// TIA Portal project "conveyer belt system V5.1" (V19)

(* hardware
DEVICE "S71500/ET200MP-Station_1"  S7-1500 station
   slot 0: "Profilschiene_0"  6ES7 590-1***0-0AA0
   slot 1: "PLC_1"  CPU 1511-1 PN  6ES7 511-1AK00-0AB0  V1.8
   slot 2: "AI 8xU/I/RTD/TC ST_1"  AI 8xU/I/RTD/TC ST  6ES7 531-7KF00-0AB0  V2.0
   slot 3: "AI 8xU/I/RTD/TC ST_2"  AI 8xU/I/RTD/TC ST  6ES7 531-7KF00-0AB0  V2.0
   slot 4: "AI 8xU/I/RTD/TC ST_3"  AI 8xU/I/RTD/TC ST  6ES7 531-7KF00-0AB0  V2.0
   slot 5: "AI 8xU/I/RTD/TC ST_4"  AI 8xU/I/RTD/TC ST  6ES7 531-7KF00-0AB0  V2.0
   slot 6: "DI 16x24VDC BA_1"  DI 16x24VDC BA  6ES7 521-1BH10-0AA0  V1.0
*)

// ===== PLC "PLC_1"  CPU 1511-1 PN =====

VAR_GLOBAL   // PLC tag table "Standard-Variablentabelle"
   "Tag_1" AT %I1000.0 : Bool;
   "Tag_2" AT %Q1000.0 : Bool;
   "Tag_3" AT %I1000.1 : Bool;
END_VAR

VAR_GLOBAL   // PLC tag table "control panel"
   "start button" AT %I0.0 : Bool;
   "reset button" AT %I0.1 : Bool;
   "stop button" AT %I0.2 : Bool;
   "emergency stop" AT %I0.3 : Bool;
   "start button light" AT %Q0.0 : Bool;
   "reset button light" AT %Q0.1 : Bool;
   "stop button light" AT %Q0.2 : Bool;
   "system start" AT %Q0.3 : Bool;
   "system fault" AT %Q0.4 : Bool;
   "system stop" AT %Q0.5 : Bool;
   "sensor start" AT %I0.7 : Bool;
   "low power mode" AT %I0.4 : Bool;
END_VAR

VAR_GLOBAL   // PLC tag table "conveyor 0"
   "motor +(0)" AT %Q3.7 : Bool;
   "motor -(0)" AT %Q3.6 : Bool;
   "encoder A(0)" AT %I3.7 : Bool;
   "encoder B(0)" AT %I3.6 : Bool;
   "sensor(0)" AT %I5.7 : Bool;
END_VAR

VAR_GLOBAL   // PLC tag table "conveyor 1"
   "motor +(1)" AT %Q3.5 : Bool;
   "motor -(1)" AT %Q3.4 : Bool;
   "encoder A(1)" AT %I3.5 : Bool;
   "encoder B(1)" AT %I3.4 : Bool;
   "sensor(1)" AT %I5.6 : Bool;
END_VAR

VAR_GLOBAL   // PLC tag table "conveyor 2"
   "motor +(2)" AT %Q3.3 : Bool;
   "motor -(2)" AT %Q3.2 : Bool;
   "encoder A(2)" AT %I3.3 : Bool;
   "encoder B(2)" AT %I3.2 : Bool;
   "sensor(2)" AT %I5.5 : Bool;
END_VAR

VAR_GLOBAL   // PLC tag table "system state"
   "start 0" AT %M0.0 : Bool;
   "start 1" AT %M0.1 : Bool;
   "conveyor 0 running" AT %M10.0 : Bool;
   "conveyor 1 running" AT %M10.1 : Bool;
   "conveyor 2 running" AT %M10.2 : Bool;
   "sensor 0 memory" AT %M20.0 : Bool;
   "sensor 1 memory" AT %M20.1 : Bool;
   "sensor 2 memory" AT %M20.2 : Bool;
   "sensor start memory" AT %M30.0 : Bool;
   "all conveyors running" AT %M0.2 : Bool;
   "system start/stop memory" AT %M0.4 : Bool;
   "conveyors running" AT %M0.3 : Bool;
   "sensor 3 memory" AT %M20.3 : Bool;
   "sensor 4 memory" AT %M20.4 : Bool;
   "sensor 5 memory" AT %M20.5 : Bool;
   "sensor 6 memory" AT %M20.6 : Bool;
   "conveyor 3 running" AT %M10.3 : Bool;
   "conveyor 4 running" AT %M10.4 : Bool;
   "conveyor 5 running" AT %M10.5 : Bool;
   "conveyor 6 running" AT %M10.6 : Bool;
END_VAR

VAR_GLOBAL   // PLC tag table "conveyor 3"
   "motor +(3)" AT %Q3.1 : Bool;
   "motor -(3)" AT %Q3.0 : Bool;
   "encoder A(3)" AT %I3.1 : Bool;
   "encoder B(3)" AT %I3.0 : Bool;
   "sensor(3)" AT %I5.4 : Bool;
END_VAR

VAR_GLOBAL   // PLC tag table "conveyor 4"
   "motor +(4)" AT %Q2.7 : Bool;
   "motor -(4)" AT %Q2.6 : Bool;
   "encoder A(4)" AT %I2.7 : Bool;
   "encoder B(4)" AT %I2.6 : Bool;
   "sensor(4)" AT %I5.3 : Bool;
END_VAR

VAR_GLOBAL   // PLC tag table "conveyor 5"
   "motor +(5)" AT %Q2.5 : Bool;
   "motor -(5)" AT %Q2.4 : Bool;
   "encoder A(5)" AT %I2.5 : Bool;
   "encoder B(5)" AT %I2.4 : Bool;
   "sensor(5)" AT %I5.2 : Bool;
END_VAR

VAR_GLOBAL   // PLC tag table "conveyor 6"
   "motor +(6)" AT %Q2.3 : Bool;
   "motor -(6)" AT %Q2.2 : Bool;
   "encoder A(6)" AT %I2.3 : Bool;
   "encoder B(6)" AT %I2.2 : Bool;
   "sensor(6)" AT %I5.1 : Bool;
END_VAR

DATA_BLOCK "conveyor_0"   // DB1
{ S7_Optimized_Access := 'TRUE' }
VERSION : 0.1
// stored: InstanceOfName conveyor control
"conveyor control"
BEGIN
END_DATA_BLOCK

DATA_BLOCK "conveyor_2"   // DB3
{ S7_Optimized_Access := 'TRUE' }
VERSION : 0.1
// stored: InstanceOfName conveyor control
"conveyor control"
BEGIN
END_DATA_BLOCK

DATA_BLOCK "conveyor_1"   // DB5
{ S7_Optimized_Access := 'TRUE' }
VERSION : 0.1
// stored: InstanceOfName conveyor control
"conveyor control"
BEGIN
END_DATA_BLOCK

DATA_BLOCK "sensor control_0"   // DB8
{ S7_Optimized_Access := 'TRUE' }
VERSION : 0.1
// stored: InstanceOfName sensor control
"sensor control"
BEGIN
END_DATA_BLOCK

DATA_BLOCK "sensor control_1"   // DB9
{ S7_Optimized_Access := 'TRUE' }
VERSION : 0.1
// stored: InstanceOfName sensor control
"sensor control"
BEGIN
END_DATA_BLOCK

DATA_BLOCK "sensor control_2"   // DB10
{ S7_Optimized_Access := 'TRUE' }
VERSION : 0.1
// stored: InstanceOfName sensor control
"sensor control"
BEGIN
END_DATA_BLOCK

DATA_BLOCK "lamp control_DB"   // DB11
{ S7_Optimized_Access := 'TRUE' }
VERSION : 0.1
// stored: InstanceOfName lamp control
"lamp control"
BEGIN
END_DATA_BLOCK

DATA_BLOCK "start pulse"   // DB12
{ S7_Optimized_Access := 'TRUE' }
VERSION : 0.1
// stored: InstanceOfName pulse
"pulse"
BEGIN
END_DATA_BLOCK

DATA_BLOCK "stop pulse"   // DB13
{ S7_Optimized_Access := 'TRUE' }
VERSION : 0.1
// stored: InstanceOfName pulse
"pulse"
BEGIN
END_DATA_BLOCK

DATA_BLOCK "conveyor_3"   // DB15
{ S7_Optimized_Access := 'TRUE' }
VERSION : 0.1
// stored: InstanceOfName conveyor control
"conveyor control"
BEGIN
END_DATA_BLOCK

DATA_BLOCK "conveyor_4"   // DB17
{ S7_Optimized_Access := 'TRUE' }
VERSION : 0.1
// stored: InstanceOfName conveyor control
"conveyor control"
BEGIN
END_DATA_BLOCK

DATA_BLOCK "conveyor_5"   // DB19
{ S7_Optimized_Access := 'TRUE' }
VERSION : 0.1
// stored: InstanceOfName conveyor control
"conveyor control"
BEGIN
END_DATA_BLOCK

DATA_BLOCK "conveyor_6"   // DB21
{ S7_Optimized_Access := 'TRUE' }
VERSION : 0.1
// stored: InstanceOfName conveyor control
"conveyor control"
BEGIN
END_DATA_BLOCK

DATA_BLOCK "sensor control_3"   // DB22
{ S7_Optimized_Access := 'TRUE' }
VERSION : 0.1
// stored: InstanceOfName sensor control
"sensor control"
BEGIN
END_DATA_BLOCK

DATA_BLOCK "sensor control_4"   // DB23
{ S7_Optimized_Access := 'TRUE' }
VERSION : 0.1
// stored: InstanceOfName sensor control
"sensor control"
BEGIN
END_DATA_BLOCK

DATA_BLOCK "sensor control_5"   // DB24
{ S7_Optimized_Access := 'TRUE' }
VERSION : 0.1
// stored: InstanceOfName sensor control
"sensor control"
BEGIN
END_DATA_BLOCK

DATA_BLOCK "sensor control_6"   // DB25
{ S7_Optimized_Access := 'TRUE' }
VERSION : 0.1
// stored: InstanceOfName sensor control
"sensor control"
BEGIN
END_DATA_BLOCK

DATA_BLOCK "standard parameters"   // DB26
{ S7_Optimized_Access := 'TRUE' }
VERSION : 0.1
   VAR
      "2 meter belt clearance delay" : Time := T#4S;
      "4 meter belt clearance delay" : Time := T#8S;
      "6 meter belt clearance delay" : Time := T#12S;
      "curved belt clearance delay" : Time := T#4S;
   END_VAR
BEGIN
END_DATA_BLOCK

DATA_BLOCK "system state"   // DB27
{ S7_Optimized_Access := 'TRUE' }
VERSION : 0.1
   VAR
      "start 0" : Bool;
      "start 1" : Bool;
      "all conveyors running" : Bool;
      "conveyors running" : Bool;
      "system start/stop memory" : Bool;
      "conveyor 0 running" : Bool;
      "conveyor 1 running" : Bool;
      "conveyor 2 running" : Bool;
      "conveyor 3 running" : Bool;
      "conveyor 4 running" : Bool;
      "conveyor 5 running" : Bool;
      "conveyor 6 running" : Bool;
      "sensor 0 memory" : Bool;
      "sensor 1 memory" : Bool;
      "sensor 2 memory" : Bool;
      "sensor 3 memory" : Bool;
      "sensor 4 memory" : Bool;
      "sensor 5 memory" : Bool;
      "sensor 6 memory" : Bool;
      "sensor start memory" : Bool;
   END_VAR
BEGIN
END_DATA_BLOCK

// folder: System blocks/Program resources

DATA_BLOCK "conveyor start delay"   // DB2
{ S7_Optimized_Access := 'TRUE' }
AUTHOR : Simatic
FAMILY : IEC
NAME : IEC_TMR
VERSION : 1.0
// stored: InstanceOfName IEC_TIMER
"IEC_TIMER"
BEGIN
END_DATA_BLOCK

DATA_BLOCK "delay 1"   // DB4
{ S7_Optimized_Access := 'TRUE' }
AUTHOR : Simatic
FAMILY : IEC
NAME : IEC_TMR
VERSION : 1.0
// stored: InstanceOfName IEC_TIMER
"IEC_TIMER"
BEGIN
END_DATA_BLOCK

DATA_BLOCK "delay 2"   // DB6
{ S7_Optimized_Access := 'TRUE' }
AUTHOR : Simatic
FAMILY : IEC
NAME : IEC_TMR
VERSION : 1.0
// stored: InstanceOfName IEC_TIMER
"IEC_TIMER"
BEGIN
END_DATA_BLOCK

DATA_BLOCK "delay 0"   // DB7
{ S7_Optimized_Access := 'TRUE' }
AUTHOR : Simatic
FAMILY : IEC
NAME : IEC_TMR
VERSION : 1.0
// stored: InstanceOfName IEC_TIMER
"IEC_TIMER"
BEGIN
END_DATA_BLOCK

DATA_BLOCK "delay 3"   // DB14
{ S7_Optimized_Access := 'TRUE' }
AUTHOR : Simatic
FAMILY : IEC
NAME : IEC_TMR
VERSION : 1.0
// stored: InstanceOfName IEC_TIMER
"IEC_TIMER"
BEGIN
END_DATA_BLOCK

DATA_BLOCK "delay 4"   // DB16
{ S7_Optimized_Access := 'TRUE' }
AUTHOR : Simatic
FAMILY : IEC
NAME : IEC_TMR
VERSION : 1.0
// stored: InstanceOfName IEC_TIMER
"IEC_TIMER"
BEGIN
END_DATA_BLOCK

DATA_BLOCK "delay 5"   // DB18
{ S7_Optimized_Access := 'TRUE' }
AUTHOR : Simatic
FAMILY : IEC
NAME : IEC_TMR
VERSION : 1.0
// stored: InstanceOfName IEC_TIMER
"IEC_TIMER"
BEGIN
END_DATA_BLOCK

DATA_BLOCK "delay 6"   // DB20
{ S7_Optimized_Access := 'TRUE' }
AUTHOR : Simatic
FAMILY : IEC
NAME : IEC_TMR
VERSION : 1.0
// stored: InstanceOfName IEC_TIMER
"IEC_TIMER"
BEGIN
END_DATA_BLOCK

// folder: (top level)

FUNCTION_BLOCK "conveyor control"   // FB1, FBD
{ S7_Optimized_Access := 'TRUE' }
VERSION : 0.1
   VAR_INPUT
      enable : Bool;
      "encoder A" : Bool;
      "encoder B" : Bool;
   END_VAR
   VAR_OUTPUT
      "running feedback" : Bool;
      "motor +" : Bool;
      "motor -" : Bool;
   END_VAR
   VAR
      "encoder buffer" : TOF_TIME;
      "encoder A edge" : R_TRIG;
      "encoder B edge" : R_TRIG;
   END_VAR
BEGIN

REGION Network 1
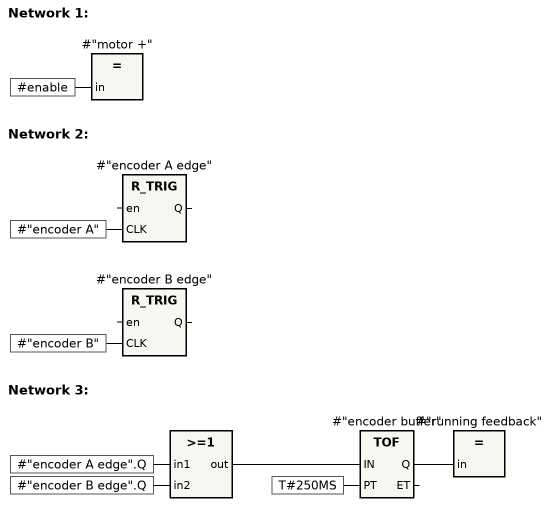
   #"motor +" := #enable;
END_REGION

REGION Network 2
   #"encoder A edge"(CLK := #"encoder A");   // R_TRIG
   #"encoder B edge"(CLK := #"encoder B");   // R_TRIG
END_REGION

REGION Network 3
   #"encoder buffer"(IN := #"encoder A edge".Q OR #"encoder B edge".Q, PT := T#250MS);   // TOF
   #"running feedback" := #"encoder buffer".Q;
END_REGION
END_FUNCTION_BLOCK

FUNCTION_BLOCK "sensor control"   // FB2, FBD
{ S7_Optimized_Access := 'TRUE' }
VERSION : 0.1
   VAR_INPUT
      "clearance delay" : Time;
      sensor : Bool;
      "preceding sensor" : Bool;
   END_VAR
   VAR_OUTPUT
      "motor +" : Bool;
   END_VAR
   VAR
      "clearance timer off" : TOF_TIME;
      "clearance timer on" : TOF_TIME;
      "clearance delay off" : TOF_TIME;
      "clearance delay on" : TON_TIME;
      "sensor memory" : Bool;
   END_VAR
BEGIN

REGION Network 1
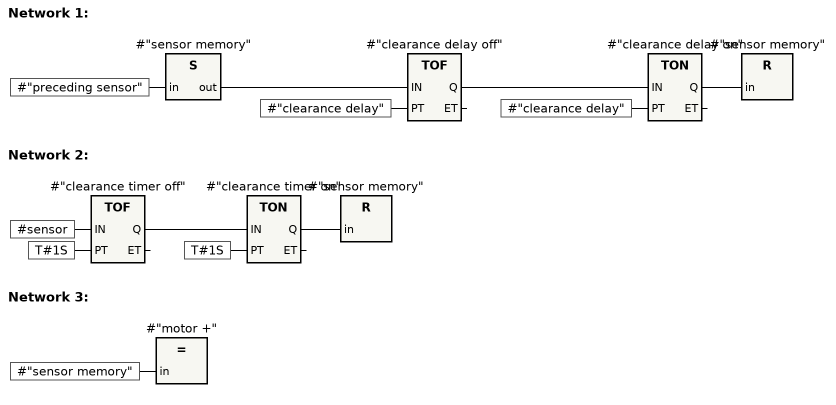
   IF #"preceding sensor" THEN #"sensor memory" := TRUE; END_IF;
   #"clearance delay off"(IN := #"preceding sensor", PT := #"clearance delay");   // TOF
   #"clearance delay on"(IN := #"clearance delay off".Q, PT := #"clearance delay");   // TON
   IF #"clearance delay on".Q THEN #"sensor memory" := FALSE; END_IF;
END_REGION

REGION Network 2
   #"clearance timer off"(IN := #sensor, PT := T#1S);   // TOF
   #"clearance timer on"(IN := #"clearance timer off".Q, PT := T#1S);   // TON
   IF #"clearance timer on".Q THEN #"sensor memory" := FALSE; END_IF;
END_REGION

REGION Network 3
   #"motor +" := #"sensor memory";
END_REGION
END_FUNCTION_BLOCK

FUNCTION_BLOCK "lamp control"   // FB3, FBD
{ S7_Optimized_Access := 'TRUE' }
VERSION : 0.1
   VAR_INPUT
      "system start" : Bool;
      "system fault" : Bool;
      "system stop" : Bool;
   END_VAR
BEGIN

REGION Network 1
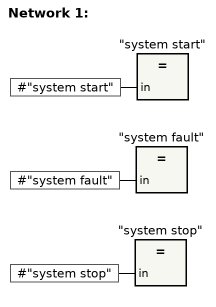
   "system start" := #"system start";
   "system fault" := #"system fault";
   "system stop" := #"system stop";
END_REGION
END_FUNCTION_BLOCK

FUNCTION_BLOCK "pulse"   // FB4, FBD
{ S7_Optimized_Access := 'TRUE' }
VERSION : 0.1
   VAR_INPUT
      enable : Bool;
      "pulse time" : Time;
   END_VAR
   VAR_OUTPUT
      "pulsing output" : Bool;
   END_VAR
   VAR
      "time delay bit" : Bool;
      IEC_Timer_0_Instance : TON_TIME;
      IEC_Timer_0_Instance_1 : TON_TIME;
   END_VAR
BEGIN

REGION Network 1
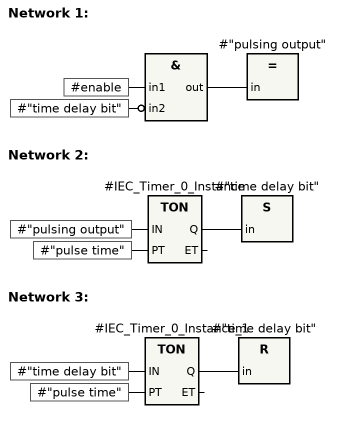
   #"pulsing output" := #enable AND NOT #"time delay bit";
END_REGION

REGION Network 2
   #IEC_Timer_0_Instance(IN := #"pulsing output", PT := #"pulse time");   // TON
   IF #IEC_Timer_0_Instance.Q THEN #"time delay bit" := TRUE; END_IF;
END_REGION

REGION Network 3
   #IEC_Timer_0_Instance_1(IN := #"time delay bit", PT := #"pulse time");   // TON
   IF #IEC_Timer_0_Instance_1.Q THEN #"time delay bit" := FALSE; END_IF;
END_REGION
END_FUNCTION_BLOCK

FUNCTION "default condition" : Void   // FC1, FBD
{ S7_Optimized_Access := 'TRUE' }
VERSION : 0.1
   VAR_TEMP   // added for the SCL form of the ladder/FBD networks
      _w1 : Bool;
      _w2 : Bool;
      _w3 : Bool;
   END_VAR
BEGIN

REGION Network 1: system start delay
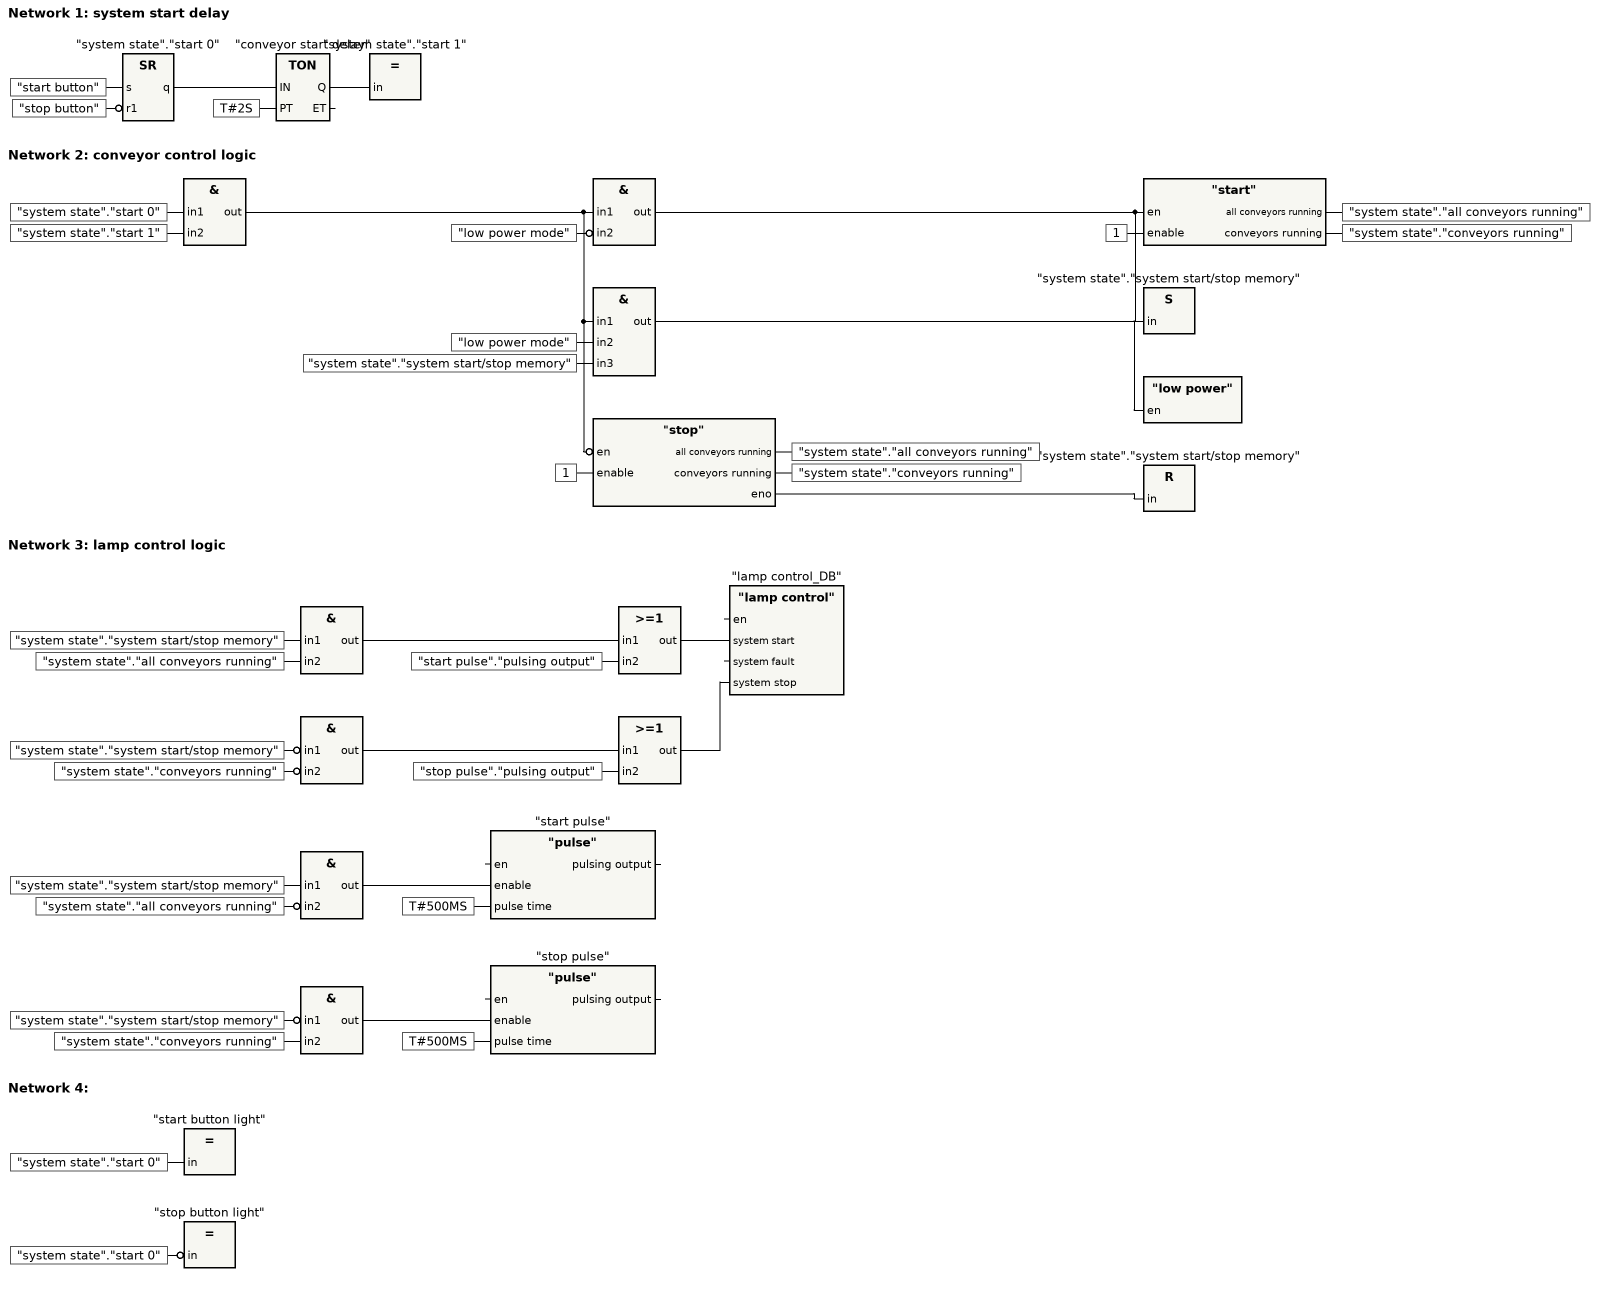
   IF "start button" THEN
       "system state"."start 0" := TRUE;   // SR flip-flop
   END_IF;
   IF NOT "stop button" THEN "system state"."start 0" := FALSE; END_IF;
   "conveyor start delay".TON(IN := "system state"."start 0", PT := T#2S);
   "system state"."start 1" := "conveyor start delay".Q;
END_REGION

REGION Network 2: conveyor control logic
   #_w1 := "system state"."start 0" AND "system state"."start 1";
   #_w2 := #_w1 AND NOT "low power mode";
   IF #_w2 THEN
       "start"(enable := 1,
               "all conveyors running" => "system state"."all conveyors running",
               "conveyors running" => "system state"."conveyors running");
       "system state"."system start/stop memory" := TRUE;
   END_IF;
   IF #_w1 AND "low power mode" AND "system state"."system start/stop memory" THEN "low power"(); END_IF;
   "stop"(EN := NOT #_w1,
          enable := 1,
          "all conveyors running" => "system state"."all conveyors running",
          "conveyors running" => "system state"."conveyors running",
          ENO => #_w3);
   IF #_w3 THEN "system state"."system start/stop memory" := FALSE; END_IF;
END_REGION

REGION Network 3: lamp control logic
   "lamp control_DB"("system start" := ("system state"."system start/stop memory" AND "system state"."all conveyors running") OR "start pulse"."pulsing output",   // "lamp control"
                     "system stop" := (NOT "system state"."system start/stop memory" AND NOT "system state"."conveyors running") OR "stop pulse"."pulsing output");
   "start pulse"(enable := "system state"."system start/stop memory" AND NOT "system state"."all conveyors running",   // "pulse"
                 "pulse time" := T#500MS);
   "stop pulse"(enable := NOT "system state"."system start/stop memory" AND "system state"."conveyors running",   // "pulse"
                "pulse time" := T#500MS);
END_REGION

REGION Network 4
   "start button light" := "system state"."start 0";
   "stop button light" := NOT "system state"."start 0";
END_REGION
END_FUNCTION

FUNCTION "start" : Void   // FC2, FBD
{ S7_Optimized_Access := 'TRUE' }
VERSION : 0.1
   VAR_INPUT
      enable : Bool;
   END_VAR
   VAR_OUTPUT
      "all conveyors running" : Bool;
      "conveyors running" : Bool;
   END_VAR
BEGIN

REGION Network 1
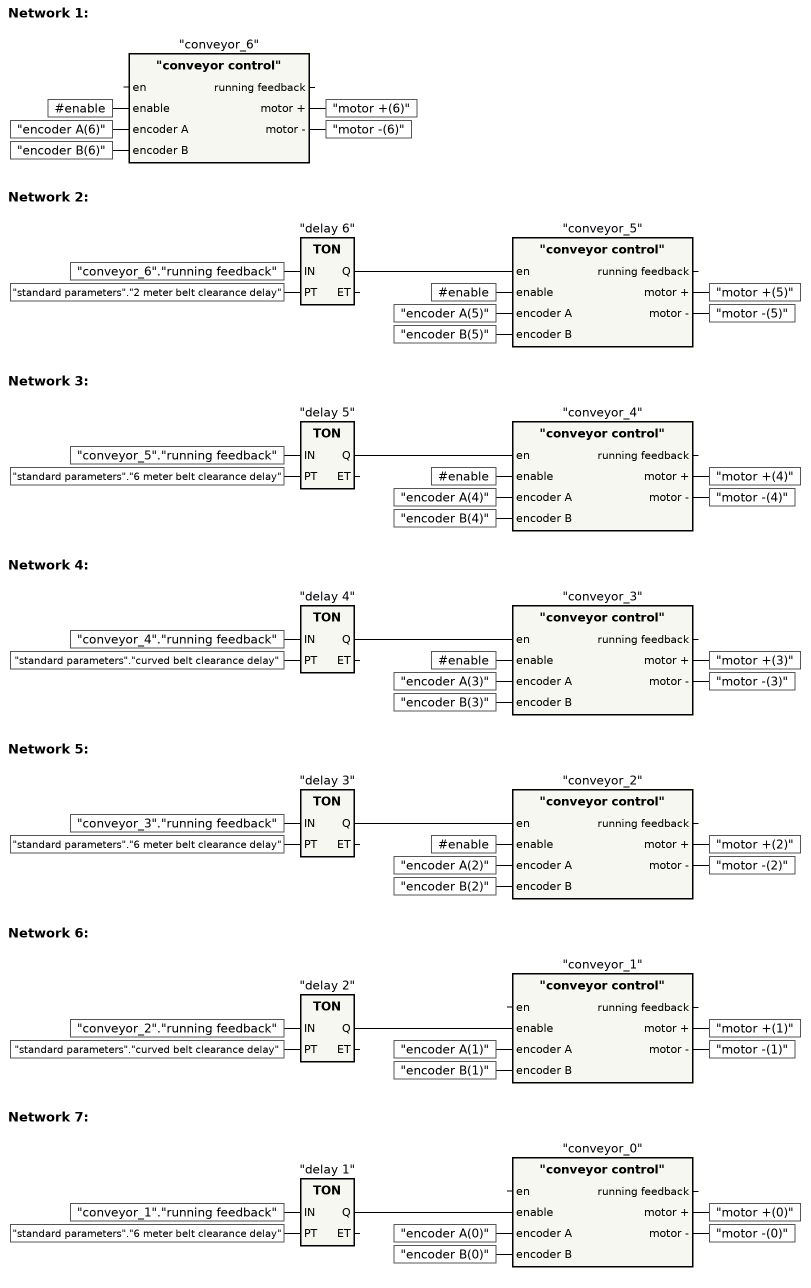
   "conveyor_6"(enable := #enable,   // "conveyor control"
                "encoder A" := "encoder A(6)",
                "encoder B" := "encoder B(6)",
                "motor +" => "motor +(6)",
                "motor -" => "motor -(6)");
END_REGION

REGION Network 2
   "delay 6".TON(IN := "conveyor_6"."running feedback",
                 PT := "standard parameters"."2 meter belt clearance delay");
   IF "delay 6".Q THEN
       "conveyor_5"(enable := #enable,   // "conveyor control"
                    "encoder A" := "encoder A(5)",
                    "encoder B" := "encoder B(5)",
                    "motor +" => "motor +(5)",
                    "motor -" => "motor -(5)");
   END_IF;
END_REGION

REGION Network 3
   "delay 5".TON(IN := "conveyor_5"."running feedback",
                 PT := "standard parameters"."6 meter belt clearance delay");
   IF "delay 5".Q THEN
       "conveyor_4"(enable := #enable,   // "conveyor control"
                    "encoder A" := "encoder A(4)",
                    "encoder B" := "encoder B(4)",
                    "motor +" => "motor +(4)",
                    "motor -" => "motor -(4)");
   END_IF;
END_REGION

REGION Network 4
   "delay 4".TON(IN := "conveyor_4"."running feedback",
                 PT := "standard parameters"."curved belt clearance delay");
   IF "delay 4".Q THEN
       "conveyor_3"(enable := #enable,   // "conveyor control"
                    "encoder A" := "encoder A(3)",
                    "encoder B" := "encoder B(3)",
                    "motor +" => "motor +(3)",
                    "motor -" => "motor -(3)");
   END_IF;
END_REGION

REGION Network 5
   "delay 3".TON(IN := "conveyor_3"."running feedback",
                 PT := "standard parameters"."6 meter belt clearance delay");
   IF "delay 3".Q THEN
       "conveyor_2"(enable := #enable,   // "conveyor control"
                    "encoder A" := "encoder A(2)",
                    "encoder B" := "encoder B(2)",
                    "motor +" => "motor +(2)",
                    "motor -" => "motor -(2)");
   END_IF;
END_REGION

REGION Network 6
   "delay 2".TON(IN := "conveyor_2"."running feedback",
                 PT := "standard parameters"."curved belt clearance delay");
   "conveyor_1"(enable := "delay 2".Q,   // "conveyor control"
                "encoder A" := "encoder A(1)",
                "encoder B" := "encoder B(1)",
                "motor +" => "motor +(1)",
                "motor -" => "motor -(1)");
END_REGION

REGION Network 7
   "delay 1".TON(IN := "conveyor_1"."running feedback",
                 PT := "standard parameters"."6 meter belt clearance delay");
   "conveyor_0"(enable := "delay 1".Q,   // "conveyor control"
                "encoder A" := "encoder A(0)",
                "encoder B" := "encoder B(0)",
                "motor +" => "motor +(0)",
                "motor -" => "motor -(0)");
END_REGION

REGION Network 8
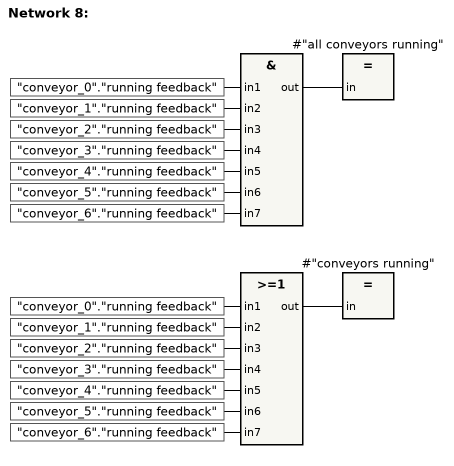
   #"all conveyors running" := "conveyor_0"."running feedback" AND "conveyor_1"."running feedback" AND "conveyor_2"."running feedback" AND "conveyor_3"."running feedback" AND "conveyor_4"."running feedback" AND "conveyor_5"."running feedback" AND "conveyor_6"."running feedback";
   #"conveyors running" := "conveyor_0"."running feedback" OR "conveyor_1"."running feedback" OR "conveyor_2"."running feedback" OR "conveyor_3"."running feedback" OR "conveyor_4"."running feedback" OR "conveyor_5"."running feedback" OR "conveyor_6"."running feedback";
END_REGION
END_FUNCTION

FUNCTION "stop" : Void   // FC3, FBD
{ S7_Optimized_Access := 'TRUE' }
VERSION : 0.1
   VAR_INPUT
      enable : Bool;
   END_VAR
   VAR_OUTPUT
      "all conveyors running" : Bool;
      "conveyors running" : Bool;
   END_VAR
BEGIN

REGION Network 1
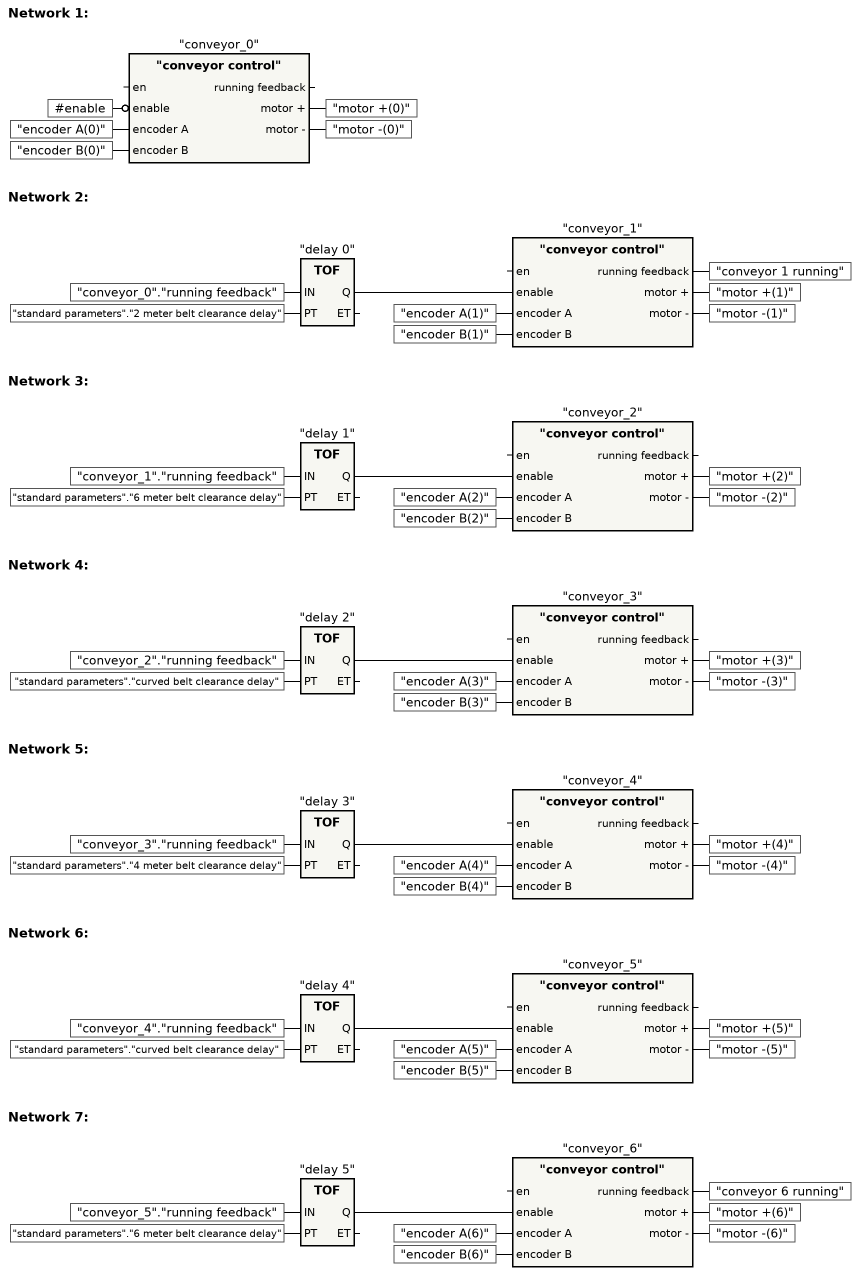
   "conveyor_0"(enable := NOT #enable,   // "conveyor control"
                "encoder A" := "encoder A(0)",
                "encoder B" := "encoder B(0)",
                "motor +" => "motor +(0)",
                "motor -" => "motor -(0)");
END_REGION

REGION Network 2
   "delay 0".TOF(IN := "conveyor_0"."running feedback",
                 PT := "standard parameters"."2 meter belt clearance delay");
   "conveyor_1"(enable := "delay 0".Q,   // "conveyor control"
                "encoder A" := "encoder A(1)",
                "encoder B" := "encoder B(1)",
                "running feedback" => "conveyor 1 running",
                "motor +" => "motor +(1)",
                "motor -" => "motor -(1)");
END_REGION

REGION Network 3
   "delay 1".TOF(IN := "conveyor_1"."running feedback",
                 PT := "standard parameters"."6 meter belt clearance delay");
   "conveyor_2"(enable := "delay 1".Q,   // "conveyor control"
                "encoder A" := "encoder A(2)",
                "encoder B" := "encoder B(2)",
                "motor +" => "motor +(2)",
                "motor -" => "motor -(2)");
END_REGION

REGION Network 4
   "delay 2".TOF(IN := "conveyor_2"."running feedback",
                 PT := "standard parameters"."curved belt clearance delay");
   "conveyor_3"(enable := "delay 2".Q,   // "conveyor control"
                "encoder A" := "encoder A(3)",
                "encoder B" := "encoder B(3)",
                "motor +" => "motor +(3)",
                "motor -" => "motor -(3)");
END_REGION

REGION Network 5
   "delay 3".TOF(IN := "conveyor_3"."running feedback",
                 PT := "standard parameters"."4 meter belt clearance delay");
   "conveyor_4"(enable := "delay 3".Q,   // "conveyor control"
                "encoder A" := "encoder A(4)",
                "encoder B" := "encoder B(4)",
                "motor +" => "motor +(4)",
                "motor -" => "motor -(4)");
END_REGION

REGION Network 6
   "delay 4".TOF(IN := "conveyor_4"."running feedback",
                 PT := "standard parameters"."curved belt clearance delay");
   "conveyor_5"(enable := "delay 4".Q,   // "conveyor control"
                "encoder A" := "encoder A(5)",
                "encoder B" := "encoder B(5)",
                "motor +" => "motor +(5)",
                "motor -" => "motor -(5)");
END_REGION

REGION Network 7
   "delay 5".TOF(IN := "conveyor_5"."running feedback",
                 PT := "standard parameters"."6 meter belt clearance delay");
   "conveyor_6"(enable := "delay 5".Q,   // "conveyor control"
                "encoder A" := "encoder A(6)",
                "encoder B" := "encoder B(6)",
                "running feedback" => "conveyor 6 running",
                "motor +" => "motor +(6)",
                "motor -" => "motor -(6)");
END_REGION

REGION Network 8
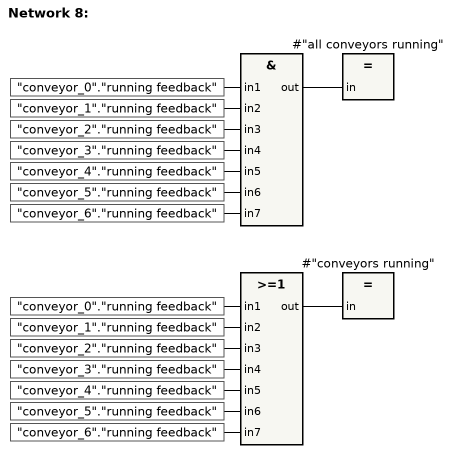
   #"all conveyors running" := "conveyor_0"."running feedback" AND "conveyor_1"."running feedback" AND "conveyor_2"."running feedback" AND "conveyor_3"."running feedback" AND "conveyor_4"."running feedback" AND "conveyor_5"."running feedback" AND "conveyor_6"."running feedback";
   #"conveyors running" := "conveyor_0"."running feedback" OR "conveyor_1"."running feedback" OR "conveyor_2"."running feedback" OR "conveyor_3"."running feedback" OR "conveyor_4"."running feedback" OR "conveyor_5"."running feedback" OR "conveyor_6"."running feedback";
END_REGION
END_FUNCTION

FUNCTION "low power" : Void   // FC4, FBD
{ S7_Optimized_Access := 'TRUE' }
VERSION : 0.1
   VAR_TEMP   // added for the SCL form of the ladder/FBD networks
      _w1 : Bool;
   END_VAR
BEGIN

REGION Network 1
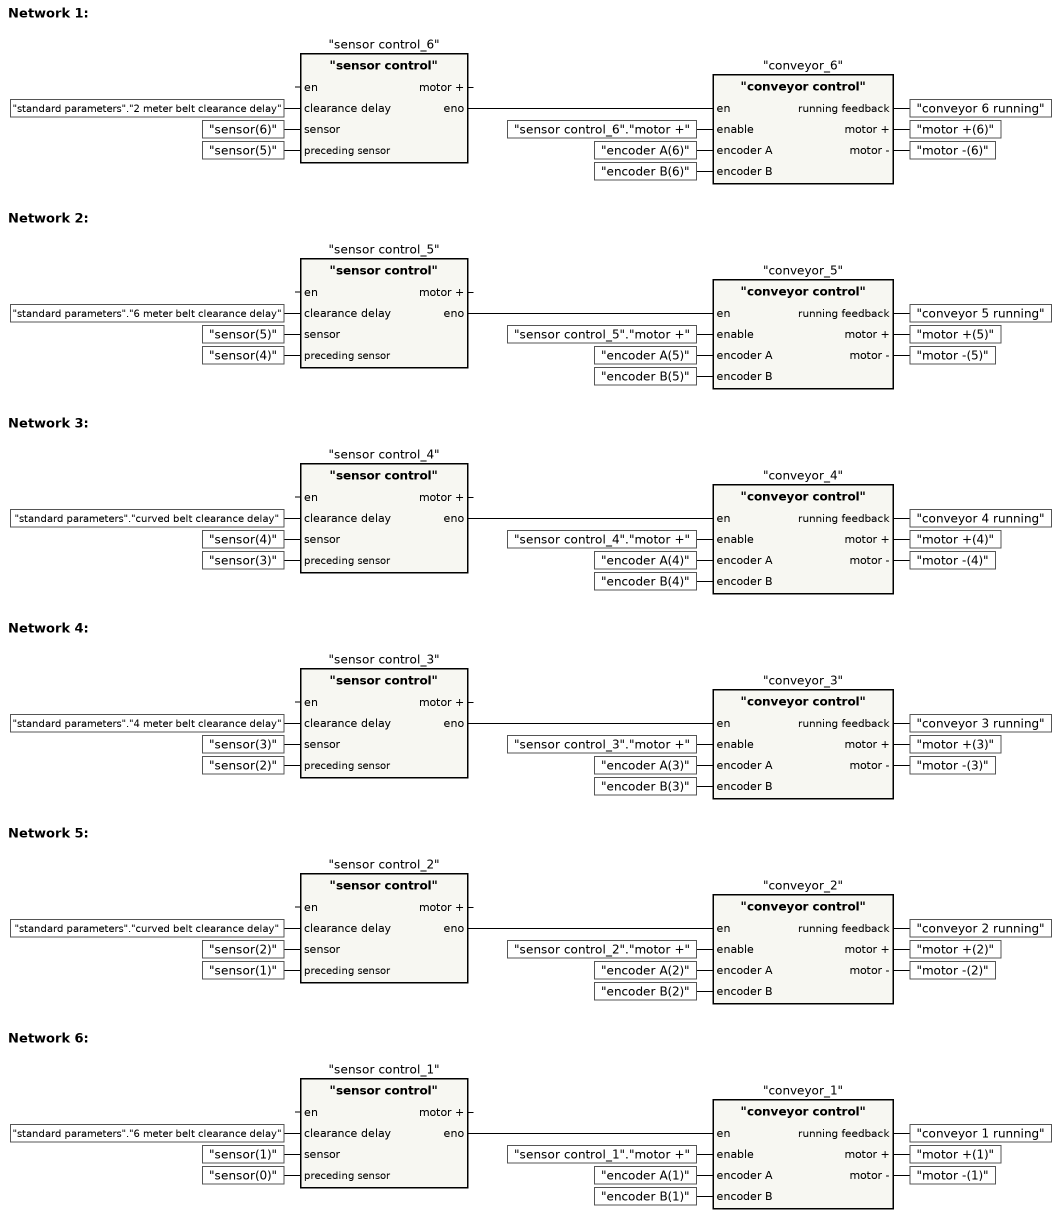
   "sensor control_6"("clearance delay" := "standard parameters"."2 meter belt clearance delay",   // "sensor control"
                      sensor := "sensor(6)",
                      "preceding sensor" := "sensor(5)",
                      ENO => #_w1);
   IF #_w1 THEN
       "conveyor_6"(enable := "sensor control_6"."motor +",   // "conveyor control"
                    "encoder A" := "encoder A(6)",
                    "encoder B" := "encoder B(6)",
                    "running feedback" => "conveyor 6 running",
                    "motor +" => "motor +(6)",
                    "motor -" => "motor -(6)");
   END_IF;
END_REGION

REGION Network 2
   "sensor control_5"("clearance delay" := "standard parameters"."6 meter belt clearance delay",   // "sensor control"
                      sensor := "sensor(5)",
                      "preceding sensor" := "sensor(4)",
                      ENO => #_w1);
   IF #_w1 THEN
       "conveyor_5"(enable := "sensor control_5"."motor +",   // "conveyor control"
                    "encoder A" := "encoder A(5)",
                    "encoder B" := "encoder B(5)",
                    "running feedback" => "conveyor 5 running",
                    "motor +" => "motor +(5)",
                    "motor -" => "motor -(5)");
   END_IF;
END_REGION

REGION Network 3
   "sensor control_4"("clearance delay" := "standard parameters"."curved belt clearance delay",   // "sensor control"
                      sensor := "sensor(4)",
                      "preceding sensor" := "sensor(3)",
                      ENO => #_w1);
   IF #_w1 THEN
       "conveyor_4"(enable := "sensor control_4"."motor +",   // "conveyor control"
                    "encoder A" := "encoder A(4)",
                    "encoder B" := "encoder B(4)",
                    "running feedback" => "conveyor 4 running",
                    "motor +" => "motor +(4)",
                    "motor -" => "motor -(4)");
   END_IF;
END_REGION

REGION Network 4
   "sensor control_3"("clearance delay" := "standard parameters"."4 meter belt clearance delay",   // "sensor control"
                      sensor := "sensor(3)",
                      "preceding sensor" := "sensor(2)",
                      ENO => #_w1);
   IF #_w1 THEN
       "conveyor_3"(enable := "sensor control_3"."motor +",   // "conveyor control"
                    "encoder A" := "encoder A(3)",
                    "encoder B" := "encoder B(3)",
                    "running feedback" => "conveyor 3 running",
                    "motor +" => "motor +(3)",
                    "motor -" => "motor -(3)");
   END_IF;
END_REGION

REGION Network 5
   "sensor control_2"("clearance delay" := "standard parameters"."curved belt clearance delay",   // "sensor control"
                      sensor := "sensor(2)",
                      "preceding sensor" := "sensor(1)",
                      ENO => #_w1);
   IF #_w1 THEN
       "conveyor_2"(enable := "sensor control_2"."motor +",   // "conveyor control"
                    "encoder A" := "encoder A(2)",
                    "encoder B" := "encoder B(2)",
                    "running feedback" => "conveyor 2 running",
                    "motor +" => "motor +(2)",
                    "motor -" => "motor -(2)");
   END_IF;
END_REGION

REGION Network 6
   "sensor control_1"("clearance delay" := "standard parameters"."6 meter belt clearance delay",   // "sensor control"
                      sensor := "sensor(1)",
                      "preceding sensor" := "sensor(0)",
                      ENO => #_w1);
   IF #_w1 THEN
       "conveyor_1"(enable := "sensor control_1"."motor +",   // "conveyor control"
                    "encoder A" := "encoder A(1)",
                    "encoder B" := "encoder B(1)",
                    "running feedback" => "conveyor 1 running",
                    "motor +" => "motor +(1)",
                    "motor -" => "motor -(1)");
   END_IF;
END_REGION

REGION Network 7
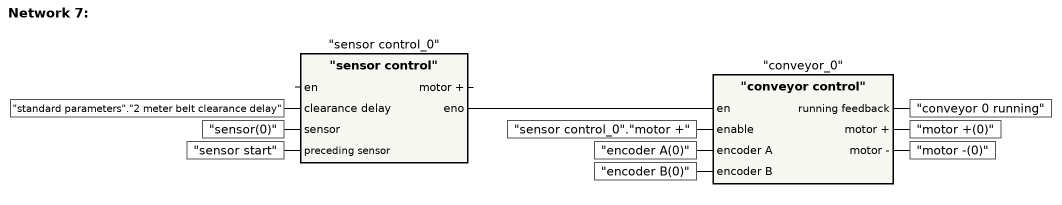
   "sensor control_0"("clearance delay" := "standard parameters"."2 meter belt clearance delay",   // "sensor control"
                      sensor := "sensor(0)",
                      "preceding sensor" := "sensor start",
                      ENO => #_w1);
   IF #_w1 THEN
       "conveyor_0"(enable := "sensor control_0"."motor +",   // "conveyor control"
                    "encoder A" := "encoder A(0)",
                    "encoder B" := "encoder B(0)",
                    "running feedback" => "conveyor 0 running",
                    "motor +" => "motor +(0)",
                    "motor -" => "motor -(0)");
   END_IF;
END_REGION
END_FUNCTION

FUNCTION "MHJ-PLC-Lab-Function-S71500" : Void   // FC9000, SCL
{ S7_Optimized_Access := 'TRUE' }
VERSION : 0.1
   VAR_TEMP
      Value : Byte;
      ForCounter : Int;
   END_VAR
   VAR CONSTANT
      Value_01_DW : DWord := 16#1223_5486;
      Value_02_DW : DWord := 16#A6C9_D1F5;
   END_VAR
BEGIN

   #Value:=PEEK(area := 16#82,
        dbNumber := 0,
        byteOffset := 511);
   #Value := #Value + 1;

   POKE(area := 16#82,
        dbNumber := 0,
        byteOffset := 511,
        value := #Value);

   POKE(area := 16#82,
        dbNumber := 0,
        byteOffset := 1016,
        value := #Value_01_DW);
   POKE(area := 16#82,
        dbNumber := 0,
        byteOffset := 1020,
        value := #Value_02_DW);

   FOR #ForCounter := 0 TO 63 DO
       #Value:=PEEK(area := 16#1,
            dbNumber := 0,
            byteOffset := #ForCounter);
       POKE(area := 16#81,
            dbNumber := 0,
            byteOffset := #ForCounter,
            value := #Value);
   END_FOR;
   #Value := PEEK(area := 16#1,
                  dbNumber := 0,
                  byteOffset := 512);
   POKE(area := 16#82,
        dbNumber := 0,
        byteOffset := 512,
        value := #Value);
END_FUNCTION

ORGANIZATION_BLOCK "Main"   // OB1, FBD, ProgramCycle
TITLE = "Main Program Sweep (Cycle)"
{ S7_Optimized_Access := 'TRUE' }
VERSION : 0.1
   VAR_INPUT
      Initial_Call : Bool;   // Initial call of this OB
      Remanence : Bool;   // =True, if remanent data are available
   END_VAR
BEGIN

REGION Network 1
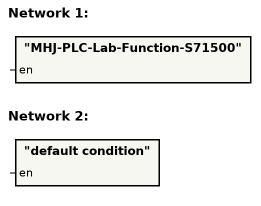
   "MHJ-PLC-Lab-Function-S71500"();
END_REGION

REGION Network 2
   "default condition"();
END_REGION
END_ORGANIZATION_BLOCK